(*
SPDX-FileCopyrightText: © 2026 Oleksandr Tiutyk <trofimich@gmail.com>
SPDX-License-Identifier: MIT
License: https://opensource.org/license/mit
*)

INTERFACE ICollectionEmptyException EXTENDS IGeneralException

METHOD Throw
VAR_INPUT
	sourceNamespaceName : STRING;
	sourceClassName : STRING;
	sourcePOUName : STRING;
	sourcePosition : STRING;
	collectionName : WSTRING;
END_VAR
END_METHOD

END_INTERFACE

(* stored: Version 1.1.0.1
   Itf ICollectionEmptyException: Id {60fb87e6-238c-4a7d-9087-bc4ff389d5a3}
   Method Throw: Id {77e34b25-d199-4c45-8866-245dc5f50505} *)
